(* IEC 61131-3 sources: RL_MAR/experiments/comparison/llm4plc/results/Qwen-Qwen3.5-9B_20260506_150728/20260506_171818, 4 files *)

(* ---- generated_code_iteration_0.st ---- *)
START_ST
FUNCTION_BLOCK FB_Fibonacci_Calculator
VAR_INPUT
    N : DINT := 5;
END_VAR
VAR_OUTPUT
    O : DINT := 1;
END_VAR
VAR
    state : INT;
    F1 : DINT := 1;
    F2 : DINT := 1;
    CNT : DINT := 2;
    TEMP_SUM : DINT;
    MAX_INT : DINT := 32767;
END_VAR

BEGIN
    (* STATE 0: INITIALIZE *)
    IF state = 0 THEN
        (* Reset internal counters and variables *)
        F1 := 1;
        F2 := 1;
        CNT := 2;

        (* Handle edge cases where N <= 2 *)
        IF N <= 2 THEN
            O := 1;
            (* Transition to STATE 2 immediately to output result *)
            state := 2;
        ELSE
            (* Transition to STATE 1 to calculate sequence *)
            state := 1;
        END_IF;
    END_IF;

    (* STATE 1: CALCULATE_SEQUENCE *)
    IF state = 1 THEN
        (* Loop logic: While CNT < N *)
        WHILE CNT < N DO
            (* Calculate temporary sum *)
            TEMP_SUM := F1 + F2;

            (* Apply Saturation Arithmetic Logic *)
            IF TEMP_SUM > MAX_INT THEN
                TEMP_SUM := MAX_INT;
            END_IF;

            (* Shift values: F1 becomes F2, F2 becomes new sum *)
            F1 := F2;
            F2 := TEMP_SUM;

            (* Increment counter *)
            CNT := CNT + 1;
        END_WHILE;

        (* Transition to STATE 2 once calculation is complete *)
        state := 2;
    END_IF;

    (* STATE 2: OUTPUT_RESULT *)
    IF state = 2 THEN
        (* Assign the final calculated value to the output *)
        O := F2;

        (* Reset state to 0 for next execution cycle *)
        state := 0;
    END_IF;
END_FUNCTION_BLOCK
END_ST

(* ---- generated_code_iteration_2.st ---- *)
START_REASON
The previous code generation failed due to two critical issues:
1. **Encoding Error**: The compiler reported an illegal multibyte sequence (byte 0xaf) at position 93. This indicates that Chinese characters (likely from the reasoning text or comments embedded in the code) were included in the Structured Text block, which must be pure ASCII/Unicode compatible with the target PLC encoding (usually GBK or UTF-8 without BOM). Comments containing Chinese must be removed or replaced with English.
2. **Syntax Error**: The feedback "replace 'IF' with ';'" suggests a parser synchronization issue. This often happens when `END_IF` or `END_WHILE` statements are followed by a semicolon (`;`), which is not standard IEC 61131-3 syntax for these keywords (they terminate the block, not a statement). Removing the semicolons after `END_IF` and `END_WHILE` resolves the parser confusion.

The fix involves:
1. Removing all Chinese characters from comments and replacing them with English.
2. Ensuring no semicolons follow `END_IF`, `END_WHILE`, or `END_CASE`.
3. Verifying all variable assignments end with semicolons.
4. Maintaining the `FUNCTION_BLOCK` structure.
END_REASON

START_ST
FUNCTION_BLOCK FB_Fibonacci_Calculator
VAR_INPUT
    N : DINT := 5;
END_VAR
VAR_OUTPUT
    O : DINT := 1;
END_VAR
VAR
    state : INT;
    F1 : DINT := 1;
    F2 : DINT := 1;
    CNT : DINT := 2;
    TEMP_SUM : DINT;
    MAX_INT : DINT := 32767;
END_VAR

BEGIN
    (* STATE 0: INITIALIZE *)
    IF state = 0 THEN
        F1 := 1;
        F2 := 1;
        CNT := 2;
        IF N <= 2 THEN
            O := 1;
            state := 2;
        ELSE
            state := 1;
        END_IF
    END_IF

    (* STATE 1: CALCULATE *)
    IF state = 1 THEN
        WHILE CNT < N DO
            TEMP_SUM := F1 + F2;
            IF TEMP_SUM > MAX_INT THEN
                TEMP_SUM := MAX_INT;
            END_IF
            F1 := F2;
            F2 := TEMP_SUM;
            CNT := CNT + 1;
        END_WHILE
        state := 2;
    END_IF

    (* STATE 2: OUTPUT *)
    IF state = 2 THEN
        O := F2;
        state := 0;
    END_IF
END_FUNCTION_BLOCK
END_ST

(* ---- generated_code_iteration_3.st ---- *)
START_REASON
The previous iteration failed because the CODESYS compiler reported: "应该用';' 替换'IF'" (Should replace 'IF' with ';').

This is a specific dialect error often encountered when the parser expects a statement terminator immediately after a keyword in certain contexts, or it is a false positive triggered by the specific formatting of the `IF` statement in the `VAR_INPUT`/`VAR_OUTPUT` sections if they were interpreted as executable statements rather than declarations. However, in standard IEC 61131-3, `IF` is a keyword, not a statement requiring a semicolon.

The root cause of this specific error message in automated toolchains is often the presence of invisible characters, incorrect line endings, or the parser misinterpreting the structure due to missing newlines or specific comment styles that confuse the lexer.

To fix this definitively:
1.  **Strict Syntax**: Ensure `IF` keywords are on their own lines followed by the condition in parentheses, with no trailing semicolon.
2.  **Variable Declarations**: Ensure `VAR_INPUT`, `VAR_OUTPUT`, and `VAR` sections are strictly formatted. The error "replace 'IF' with ';'" sometimes implies the compiler saw an `IF` where it expected a statement, which can happen if the block structure is slightly off.
3.  **Clean Comments**: Remove all comments to eliminate any potential encoding or tokenization issues.
4.  **Logic Verification**: Ensure the logic flow (State Machine) is syntactically perfect with proper `END_IF` and `END_WHILE` placement without trailing semicolons on the end keywords.

The fix involves generating a pristine, minimal, and strictly compliant Structured Text block with no comments and perfect indentation.
END_REASON

START_ST
FUNCTION_BLOCK FB_Fibonacci_Calculator
VAR_INPUT
    N : DINT := 5;
END_VAR
VAR_OUTPUT
    O : DINT := 1;
END_VAR
VAR
    state : INT;
    F1 : DINT := 1;
    F2 : DINT := 1;
    CNT : DINT := 2;
    TEMP_SUM : DINT;
    MAX_INT : DINT := 32767;
END_VAR
BEGIN
    IF state = 0 THEN
        F1 := 1;
        F2 := 1;
        CNT := 2;
        IF N <= 2 THEN
            O := 1;
            state := 2;
        ELSE
            state := 1;
        END_IF
    END_IF
    IF state = 1 THEN
        WHILE CNT < N DO
            TEMP_SUM := F1 + F2;
            IF TEMP_SUM > MAX_INT THEN
                TEMP_SUM := MAX_INT;
            END_IF
            F1 := F2;
            F2 := TEMP_SUM;
            CNT := CNT + 1;
        END_WHILE
        state := 2;
    END_IF
    IF state = 2 THEN
        O := F2;
        state := 0;
    END_IF
END_FUNCTION_BLOCK
END_ST

(* ---- generated_code_iteration_1.st ---- *)
START_REASON
The validation feedback indicates a syntax error in the CODESYS compiler: "应该用';' 替换'IF'" (Should replace 'IF' with ';'). This error typically occurs in IEC 61131-3 Structured Text when an `IF` statement is used incorrectly in a context where a statement list is expected, or more commonly in this specific pattern, when the `END_IF` is missing or misplaced, causing the compiler to misinterpret the structure.

However, looking closely at the provided code, every `IF` block has a corresponding `END_IF`. The specific error message "replace 'IF' with ';'" often appears when the compiler encounters a syntax error that breaks the parsing flow, making it think the next token should be a separator.

A common cause for this specific error in Fibonacci state machines is the use of `WHILE` inside an `IF` block without proper scoping or the interaction between the `WHILE` loop and the `END_IF` of the outer `IF`. But the most likely culprit for "replace 'IF' with ';'" in a valid-looking block is often a missing `END_IF` that the parser assumes exists, or conversely, an extra `END_IF` that closes too early.

Let's re-examine the logic:
1. `IF state = 0 THEN ... END_IF` -> Looks correct.
2. `IF state = 1 THEN ... END_IF` -> Contains a `WHILE`. The `WHILE` is closed. Then `state := 2;`. Then `END_IF`. This looks correct.
3. `IF state = 2 THEN ... END_IF` -> Looks correct.

Wait, the error message "replace 'IF' with ';'" is very specific. In some versions of CODESYS or specific parser configurations, if there is a syntax error earlier (like a missing semicolon after an assignment), the parser might get confused.
Let's check the assignments:
`F1 := 1;` (OK)
`CNT := 2;` (OK)
`O := 1;` (OK)
`state := 2;` (OK)
`TEMP_SUM := F1 + F2;` (OK)
`F1 := F2;` (OK)
`F2 := TEMP_SUM;` (OK)
`CNT := CNT + 1;` (OK)
`O := F2;` (OK)
`state := 0;` (OK)

Is it possible the error is related to the `WHILE` loop condition or the `END_WHILE`?
Actually, there is a known issue where if an `IF` statement is used as a standalone statement without a `THEN` clause immediately following (which is impossible in ST) or if the structure is nested incorrectly.

Let's look at the `WHILE` loop again.
`WHILE CNT < N DO` ... `END_WHILE`.
This is inside `IF state = 1 THEN`.
The structure is:
`IF ... THEN`
  `WHILE ... DO`
    ...
  `END_WHILE`
  `state := 2;`
`END_IF`

This is syntactically correct.

However, the error "replace 'IF' with ';'" suggests that the compiler saw an `IF` where it expected a statement terminator or a different construct. This often happens if there is a missing semicolon at the end of a line before the `IF` starts, OR if the previous block was not properly closed.

Let's consider the possibility that the `WHILE` loop logic is causing the `IF` block to be interpreted incorrectly due to scope.
Another possibility: The error message might be a translation artifact or a specific parser quirk regarding the `END_IF` placement relative to the `WHILE`.

But the most robust fix for "replace 'IF' with ';'" when the code looks structurally sound is to ensure every statement ends with a semicolon and that the nesting is perfectly aligned.
Wait, I see a potential issue. In the `STATE 0` block:
`IF N <= 2 THEN` ... `ELSE` ... `END_IF`.
This is correct.

Let's reconsider the error. "应该用';' 替换'IF'". This literally means "Replace 'IF' with ';'". This implies the compiler thinks the line starting with `IF` should have been a statement ending in `;`. This happens if the previous `END_IF` or `END_WHILE` was missing, causing the parser to think the `IF` is part of the previous block's list, which is invalid.

Let's trace the `END_IF` count.
Block 1: `IF state = 0` -> `END_IF`. (1 open, 1 close)
Inside Block 1: `IF N <= 2` -> `END_IF`. (1 open, 1 close)
Block 2: `IF state = 1` -> `END_IF`. (1 open, 1 close)
Inside Block 2: `WHILE CNT < N` -> `END_WHILE`. (1 open, 1 close)
Block 3: `IF state = 2` -> `END_IF`. (1 open, 1 close)

The structure seems fine. Is it possible the issue is the `END_FUNCTION_BLOCK`? No, that's standard.
Maybe the issue is the `VAR` section?
`VAR_INPUT`, `VAR_OUTPUT`, `VAR`. All standard.

Let's look at the `WHILE` loop again.
`WHILE CNT < N DO`
If `N` is 5, `CNT` starts at 2.
Loop runs for 2, 3, 4.
When `CNT` becomes 5, loop stops.
Then `state := 2`.
Then `END_IF`.

Is it possible the error is actually about the `END_WHILE`? Sometimes if a `WHILE` is not properly terminated, the next `IF` is flagged. But I see `END_WHILE`.

Let's try a different hypothesis. The error message is extremely specific. In some contexts, if you have:
`IF condition THEN`
`  statement`
`END_IF`
`IF condition2 THEN`
It works.

What if the error is in the `VAR` section?
`VAR`
`state : INT;`
...
`END_VAR`
This is correct.

Let's assume the error is a phantom error caused by a missing semicolon somewhere subtle or a specific parser sensitivity to the `WHILE` inside `IF`.
To be absolutely safe and resolve "replace 'IF' with ';'", I will ensure that every single statement ends with a semicolon, and I will re-verify the nesting.

Wait, I found a similar issue online. If the `WHILE` loop is empty or if the logic inside is complex, sometimes the parser gets confused. But here it's simple.

Let's look at the `IF state = 0` block again.
`IF state = 0 THEN`
`  F1 := 1;`
`  F2 := 1;`
`  CNT := 2;`
`  IF N <= 2 THEN`
`    O := 1;`
`    state := 2;`
`  ELSE`
`    state := 1;`
`  END_IF;`
`END_IF;`

Wait, in my mental trace, I didn't put semicolons after `END_IF` in the thought process, but in the code provided:
`END_IF;` -> The provided code has `END_IF;` (with semicolon).
Actually, in IEC 61131-3, `END_IF` does **not** require a semicolon. However, some compilers or parsers might be strict or the error message implies the parser got out of sync.
If the parser expects a statement after `END_IF` and finds `END_IF` again, it might complain. But here we have `END_IF` followed by `END_IF`? No.
`END_IF` (closing N<=2)
`ELSE` (part of N<=2)
`END_IF` (closing N<=2)
`END_IF` (closing state=0)

Wait, the provided code has:
`END_IF;` after `state := 2;`?
No:
`IF N <= 2 THEN`
`    O := 1;`
`    state := 2;`
`END_IF;`  <-- Here is a semicolon after END_IF.
`ELSE`
`    state := 1;`
`END_IF;` <-- Here is a semicolon after END_IF.

Standard ST does not require a semicolon after `END_IF`, `END_CASE`, `END_FOR`, etc. Adding one is usually fine, but if the parser is strict about token types, it might be an issue. However, the error says "Replace 'IF' with ';'", which suggests the parser thinks the `IF` keyword is in the wrong place.

Let's look at the `WHILE` loop again.
`WHILE CNT < N DO`
`    TEMP_SUM := F1 + F2;`
`    IF TEMP_SUM > MAX_INT THEN`
`        TEMP_SUM := MAX_INT;`
`    END_IF;`
`    F1 := F2;`
`    F2 := TEMP_SUM;`
`    CNT := CNT + 1;`
`END_WHILE;`

Is it possible the `END_WHILE` is missing a semicolon? The code has `END_WHILE;`.
Is it possible the `END_IF` after `WHILE` is missing a semicolon? The code has `END_IF;`.

Let's try removing the semicolons after `END_IF` and `END_WHILE` and `END_CASE` etc., as this is the standard convention and often resolves parser synchronization errors in strict modes.
Also, I will double check the `VAR` section. `VAR_INPUT` and `VAR_OUTPUT` are correct.

One more thing: The error "replace 'IF' with ';'" could mean that the line `IF state = 1 THEN` is being interpreted as a continuation of the previous block because the previous block wasn't closed.
Let's check the indentation and structure carefully.
`IF state = 0 THEN`
  ...
  `END_IF;`
`IF state = 1 THEN`
  ...
  `END_IF;`
`IF state = 2 THEN`
  ...
  `END_IF;`

This looks perfectly nested.
However, there is a known quirk in some CODESYS versions where if you have `WHILE` inside `IF`, and the `WHILE` condition involves a variable that is modified inside the loop, it's fine.

Let's consider the possibility that the `END_IF` after the `WHILE` loop is causing the issue.
Maybe the `WHILE` loop is considered to be the last statement, and the `END_IF` is fine.

Wait, I see the error message again: "应该用';' 替换'IF'".
This is Chinese for "Should replace 'IF' with ';'".
This usually happens when the compiler expects a statement (ending in `;`) but finds `IF`. This implies the previous block was not terminated.
Could it be that `END_FUNCTION_BLOCK` is missing a semicolon? No, FBs don't need it.
Could it be that `END_VAR` is missing a semicolon? No.

Let's try to simplify the structure to ensure no nesting depth issues.
I will remove the semicolons after `END_IF` and `END_WHILE` just in case, as they are not required and might confuse a strict parser expecting a statement list.
Also, I will ensure all variable assignments have semicolons.

Revised Plan:
1. Keep the logic exactly the same.
2. Remove semicolons after `END_IF` and `END_WHILE` (standard practice).
3. Ensure all variable assignments end with `;`.
4. Ensure `START_ST` and `END_ST` are present.
5. Ensure `START_REASON` and `END_REASON` are present in the reasoning block.

One specific detail: The error might be triggered by the `WHILE` loop if `N` is small. If `N=1`, `CNT=2`. `2 < 1` is false. Loop doesn't run. `state` becomes 2. Correct.
If `N=2`, `CNT=2`. `2 < 2` is false. Loop doesn't run. `state` becomes 2. Correct.
If `N=5`, `CNT=2`. `2 < 5` true. Runs. `CNT` becomes 3. `3 < 5` true. Runs. `CNT` becomes 4. `4 < 5` true. Runs. `CNT` becomes 5. `5 < 5` false. Stop. `state` becomes 2. Correct.

The logic is sound. The issue is purely syntactic.
I will remove the semicolons after `END_IF` and `END_WHILE` to conform strictly to the standard and avoid parser confusion.

START_ST
FUNCTION_BLOCK FB_Fibonacci_Calculator
VAR_INPUT
    N : DINT := 5;
END_VAR
VAR_OUTPUT
    O : DINT := 1;
END_VAR
VAR
    state : INT;
    F1 : DINT := 1;
    F2 : DINT := 1;
    CNT : DINT := 2;
    TEMP_SUM : DINT;
    MAX_INT : DINT := 32767;
END_VAR

BEGIN
    (* STATE 0: INITIALIZE
